(* PLC project model_InDecode, Beckhoff Automation Beckhoff MLlib 3.1.251201.0 *)
(* stored: creationDateTime 2026-06-04T05:12:43.2676280, modificationDateTime 2026-06-04T05:12:43.2676280 *)

TYPE ST_model_InDecodeInput :
STRUCT

	{attribute 'hide'} _header_DO_NOT_CHANGE : ARRAY[0..63] OF SINT := [-1,-112,120,86,52,18,-1,-1,1,-1,0,0,-1,-1,-112,-112,-98,30,108,37,-121,74,-126,76,-75,77,-89,33,-107,61,4,-86,-123,62,115,41,123,-85,-72,-46,-70,-45,0,87,2,-106,-29,-87,64,0,75,0,0,0,0,0,0,0,0,0,0,0,0,0];
	in_images : ARRAY[0..0,0..2,0..639,0..639] OF REAL;

END_STRUCT
END_TYPE

TYPE ST_model_InDecodeOutput :
STRUCT

	{attribute 'hide'} _header_DO_NOT_CHANGE : ARRAY[0..63] OF SINT := [-1,-112,120,86,52,18,-1,-1,1,-1,0,0,-1,-1,-112,-112,-97,-47,126,-66,90,56,100,-109,-99,-74,-40,-64,48,11,33,45,-41,-24,68,80,115,94,-74,-30,85,-101,111,-94,20,-24,42,26,-64,19,3,0,0,0,0,0,0,0,0,0,0,0,0,0];
	out_output : ARRAY[0..0,0..8399,0..5] OF REAL;

END_STRUCT
END_TYPE
